// TIA Portal project "Project11" (V19)

(* hardware
DEVICE "S7-1500/ET200MP station_1"  S7-1500 station
   slot 0: "Rail_0"  Rack  6ES7 590-1***0-0AA0
   slot 1: "PLC_1"  CPU 1511-1 PN  6ES7 511-1AK02-0AB0  V2.9
      slot 3: "CPU display_1"  6ES7591-1AA00-0AA0
      slot 32768: "PROFINET interface_1"  X1
         slot 32769: "Port_1"  X1 P1
         slot 32770: "Port_2"  X1 P2
      slot 34817: "Virtual CP interface port_1"  Virtual CP interface port  Virtual CP interface port
   slot 2: "CM 1542-1_1"  CM 1542-1  6GK7 542-1AX00-0XE0  V3.0
   slot 3: "CP 1543-1_1"  CP 1543-1  6GK7 543-1AX00-0XE0  V3.0
DEVICE "HMI_1"  TP700 Comfort
   slot 0: "HMI_1"  TP700 Comfort  6AV2 124-0GC01-0AX0  17.0.0.0
   slot 1: "HMI_RT_1"  TP700 Comfort  6AV2 124-0GC01-0AX0  17.0.0.0
   slot 5: "HMI_1.IE_CP_1"  PROFINET Interface  17.0.0.0
      slot 1: "PROFINET Interface_1"  PROFINET Interface
         slot 1: "Port_1"  Port
         slot 2: "Port_2"  Port
   slot 7: "HMI_1.MPI/DP_CP_1"  MPI/DP Interface  17.0.0.0
DEVICE "HMI_2"  TP700 Comfort
   slot 0: "HMI_2"  TP700 Comfort  6AV2 124-0GC01-0AX0  17.0.0.0
   slot 1: "HMI_RT_2"  TP700 Comfort  6AV2 124-0GC01-0AX0  17.0.0.0
   slot 5: "HMI_2.IE_CP_1"  PROFINET Interface  17.0.0.0
      slot 1: "PROFINET Interface_1"  PROFINET Interface
         slot 1: "Port_1"  Port
         slot 2: "Port_2"  Port
   slot 7: "HMI_2.MPI/DP_CP_1"  MPI/DP Interface  17.0.0.0
DEVICE "HMI_3"  TP700 Comfort
   slot 0: "HMI_3"  TP700 Comfort  6AV2 124-0GC01-0AX0  17.0.0.0
   slot 1: "HMI_RT_3"  TP700 Comfort  6AV2 124-0GC01-0AX0  17.0.0.0
   slot 5: "HMI_3.IE_CP_1"  PROFINET Interface  17.0.0.0
      slot 1: "PROFINET Interface_1"  PROFINET Interface
         slot 1: "Port_1"  Port
         slot 2: "Port_2"  Port
   slot 7: "HMI_3.MPI/DP_CP_1"  MPI/DP Interface  17.0.0.0
*)

// ===== PLC "PLC_1"  CPU 1511-1 PN =====

VAR_GLOBAL   // PLC tag table "Tag table_1"
   "HMI_1" AT %M0.0 : Bool;
   "HMI_2" AT %M0.1 : Bool;
   "HMI_3" AT %M0.2 : Bool;
END_VAR

ORGANIZATION_BLOCK "Main"   // OB1, LAD, ProgramCycle
TITLE = "Main Program Sweep (Cycle)"
{ S7_Optimized_Access := 'TRUE' }
VERSION : 0.1
   VAR_INPUT
      Initial_Call : Bool;   // Initial call of this OB
      Remanence : Bool;   // =True, if remanent data are available
   END_VAR
BEGIN

REGION Network 1
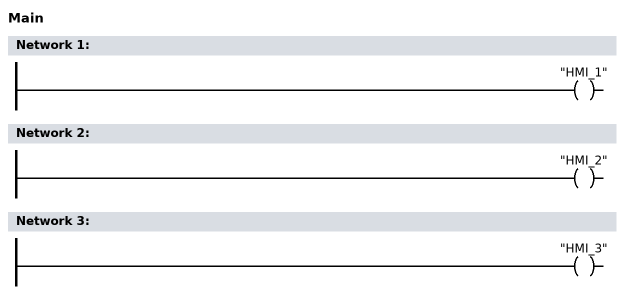
   RUNG wire#powerrail
      Coil( "HMI_1" )
   END_RUNG
   // the same network as SCL:
   "HMI_1" := TRUE;
END_REGION

REGION Network 2
   RUNG wire#powerrail
      Coil( "HMI_2" )
   END_RUNG
   // the same network as SCL:
   "HMI_2" := TRUE;
END_REGION

REGION Network 3
   RUNG wire#powerrail
      Coil( "HMI_3" )
   END_RUNG
   // the same network as SCL:
   "HMI_3" := TRUE;
END_REGION
END_ORGANIZATION_BLOCK

(* ===== HMI "HMI_RT_1" =====
connection "HMI_Connection_1": ETHERNET, S7_1500_OMS

HMI tags "Default tag table"
   "HMI_1" : Bool = PLC HMI_1 AT %M0.0, 1 s

screen "Screen_1" 800x480
   IOField "I/O field_1" at 301,143 size 96x32; FormatPattern 1
      ProcessValue <- "HMI_1"
*)

(* ===== HMI "HMI_RT_2" =====
connection "HMI_Connection_2": ETHERNET, S7_1500_OMS

HMI tags "Default tag table"
   "HMI_2" : Bool = PLC HMI_2 AT %M0.1, 1 s

screen "Screen_1" 800x480
   IOField "I/O field_1" at 317,163 size 96x32; FormatPattern 1
      ProcessValue <- "HMI_2"
*)

(* ===== HMI "HMI_RT_3" =====
connection "HMI_Connection_3": ETHERNET, S7_1500_OMS

HMI tags "Default tag table"
   "HMI_3" : Bool = PLC HMI_3 AT %M0.2, 1 s

screen "Screen_1" 800x480
   IOField "I/O field_1" at 180,214 size 96x32; FormatPattern 1
      ProcessValue <- "HMI_3"
*)